Xinje XDPPro project, PLC1: XDC-60C4 (software 3.3 2016-01-26 内部测试:短信配置，自由格式配置)

PROGRAM Ladder

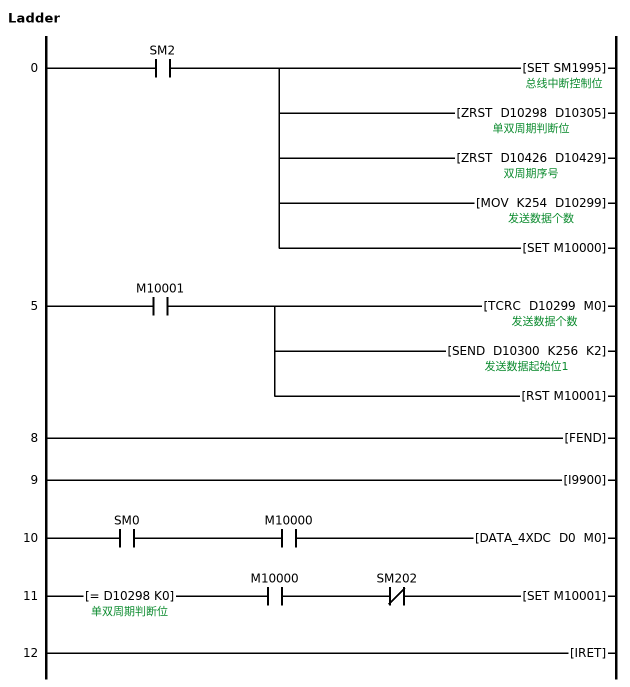
LD     SM2
SET    SM1995	; 总线中断控制位
ZRST   D10298 D10305	; 单双周期判断位
ZRST   D10426 D10429	; 双周期序号
MOV    K254 D10299	; 发送数据个数
SET    M10000
LD     M10001
TCRC   D10299 M0	; 发送数据个数
SEND   D10300 K256 K2	; 发送数据起始位1
RST    M10001
FEND
I9900
LD     SM0
AND    M10000
DATA_4XDC D0 M0
LD=    D10298 K0	; 单双周期判断位
AND    M10000
ANI    SM202
SET    M10001
IRET

COMMENTS (devices not used above)
D10301	发送数据起始位2
D10302	单周期序号
D10400	双周期数据起始位
D10554	CRC校验位
D10555	CRC校验位

C FUNCTION BLOCK data_4xdc.fcb
/*************************************************************************
   FunctionBlockName:  DATA_4XDC
   Version:            1.0.0
   Author:             cxw
   UpdateTime:         2016-1-22 15:31:37
   Comment:            
			
**************************************************************************/
void DATA_4XDC( WORD W , BIT B )
{
	#define SysRegAddr_HD_D_SD_HSD_SM
	#define offset 10300			//偏移量
	
	int i=0,j=0;
	INT16U sign=0x00ff;
	
	D[offset+0] = 0x0055;			//起始符1
	D[offset+1] = 0x0055;			//起始符2
	
	if(D[offset-2] == 0)					//单双周期判断
	{
		D[offset+2] = D[offset+126]+1;		//上周期数据序号						
		D[offset+3] = D[offset+127];
		D[offset+4] = D[offset+128];
		D[offset+5] = D[offset+129];
		
		for(i=0,j=0;i<3;i=i+1)		//轴1~3
		{
			j = i;
			D[offset+6+40*j] = (*(INT16S*)&HSD[100+20*i]&0x00ff);		//轴1位置给定
			D[offset+7+40*j] = (*(INT16S*)&HSD[100+20*i]&0xff00)>>8;
			D[offset+8+40*j] = (*(INT16S*)&HSD[101+20*i]&0x00ff);
			D[offset+9+40*j] = (*(INT16S*)&HSD[101+20*i]&0xff00)>>8;
			D[offset+10+40*j] = (*(INT16S*)&HSD[104+20*i]&0x00ff);		//轴1位置反馈
			D[offset+11+40*j] = (*(INT16S*)&HSD[104+20*i]&0xff00)>>8;
			D[offset+12+40*j] = (*(INT16S*)&HSD[105+20*i]&0x00ff);
			D[offset+13+40*j] = (*(INT16S*)&HSD[105+20*i]&0xff00)>>8;
			D[offset+14+40*j] = (*(INT16S*)&HSD[108+20*i]&0x00ff);		//轴1当前次位移脉冲数
			D[offset+15+40*j] = (*(INT16S*)&HSD[108+20*i]&0xff00)>>8;
			D[offset+16+40*j] = (*(INT16S*)&HSD[109+20*i]&0x00ff);
			D[offset+17+40*j] = (*(INT16S*)&HSD[109+20*i]&0xff00)>>8;
			
			D[offset+18+40*j] = (*(INT16S*)&SD[2012+60*i]&0x00ff);		//轴1瞬时速度给定
			D[offset+19+40*j] = (*(INT16S*)&SD[2012+60*i]&0xff00)>>8;
			D[offset+20+40*j] = (*(INT16S*)&SD[2013+60*i]&0x00ff);
			D[offset+21+40*j] = (*(INT16S*)&SD[2013+60*i]&0xff00)>>8;
			D[offset+22+40*j] = (*(INT16S*)&SD[2030+60*i]&0x00ff);		//轴1位置设定
			D[offset+23+40*j] = (*(INT16S*)&SD[2030+60*i]&0xff00)>>8;
			D[offset+24+40*j] = (*(INT16S*)&SD[2031+60*i]&0x00ff);
			D[offset+25+40*j] = (*(INT16S*)&SD[2031+60*i]&0xff00)>>8;
			D[offset+26+40*j] = (*(INT16S*)&SD[2032+60*i]&0x00ff);		//轴1速度设定
			D[offset+27+40*j] = (*(INT16S*)&SD[2032+60*i]&0xff00)>>8;
			D[offset+28+40*j] = (*(INT16S*)&SD[2033+60*i]&0x00ff);
			D[offset+29+40*j] = (*(INT16S*)&SD[2033+60*i]&0xff00)>>8;
			D[offset+30+40*j] = (*(INT16S*)&SD[2034+60*i]&0x00ff);		//轴1加速时间
			D[offset+31+40*j] = (*(INT16S*)&SD[2034+60*i]&0xff00)>>8;
			D[offset+32+40*j] = (*(INT16S*)&SD[2035+60*i]&0x00ff);					
			D[offset+33+40*j] = (*(INT16S*)&SD[2035+60*i]&0xff00)>>8;
			D[offset+34+40*j] = (*(INT16S*)&SD[2036+60*i]&0x00ff);		//轴1减速时间
			D[offset+35+40*j] = (*(INT16S*)&SD[2036+60*i]&0xff00)>>8;
			D[offset+36+40*j] = (*(INT16S*)&SD[2037+60*i]&0x00ff);					
			D[offset+37+40*j] = (*(INT16S*)&SD[2037+60*i]&0xff00)>>8;
			D[offset+38+40*j] = (*(INT16S*)&SD[2002+60*i]&0x00ff);		//轴1错误代码
			D[offset+39+40*j] = (*(INT16S*)&SD[2003+60*i]&0xff00)>>8;
			
			D[offset+40+40*j] = ((INT16U)SM[2000+20*i]);				//轴1使能标志
			D[offset+41+40*j] = ((INT16U)SM[2001+20*i]);				//轴1正在运动标志
			D[offset+42+40*j] = ((INT16U)SM[2003+20*i]);				//轴1指令完成标志
			D[offset+43+40*j] = ((INT16U)SM[2004+20*i]);				//轴1错误标志
			D[offset+44+40*j] = ((INT16U)SM[2010+20*i]);				//轴1使能控制位
			D[offset+45+40*j] = sign;
		}
		D[offset-2] = D[offset-2]+1;			
	}
	else
	{
		D[offset+126] = D[offset+2]+1;			//上周期数据序号
		if(D[offset+126]>=256)
		{
			D[offset+126] = 0;
			D[offset+127] = D[offset+127]+1;
		}
		if(D[offset+127]>=256)
		{
			D[offset+127] = 0;
			D[offset+128] = D[offset+128]+1;
		}
		if(D[offset+128]>=256)
		{
			D[offset+128] = 0;
			D[offset+129] = D[offset+129]+1;
		}
		if(D[offset+129]>=256)
		{
			D[offset+129] = 0;
		}
		
		for(i=0,j=0;i<3;i++)
		{
			j = i;
			D[offset+130+40*j] = (*(INT16S*)&HSD[100+20*i]&0x00ff);		//轴1位置给定
			D[offset+131+40*j] = (*(INT16S*)&HSD[100+20*i]&0xff00)>>8;
			D[offset+132+40*j] = (*(INT16S*)&HSD[101+20*i]&0x00ff);
			D[offset+133+40*j] = (*(INT16S*)&HSD[101+20*i]&0xff00)>>8;
			D[offset+134+40*j] = (*(INT16S*)&HSD[104+20*i]&0x00ff);		//轴1位置反馈
			D[offset+135+40*j] = (*(INT16S*)&HSD[104+20*i]&0xff00)>>8;
			D[offset+136+40*j] = (*(INT16S*)&HSD[105+20*i]&0x00ff);
			D[offset+137+40*j] = (*(INT16S*)&HSD[105+20*i]&0xff00)>>8;
			D[offset+138+40*j] = (*(INT16S*)&HSD[108+20*i]&0x00ff);		//轴1当前次位移脉冲数
			D[offset+139+40*j] = (*(INT16S*)&HSD[108+20*i]&0xff00)>>8;
			D[offset+140+40*j] = (*(INT16S*)&HSD[109+20*i]&0x00ff);
			D[offset+141+40*j] = (*(INT16S*)&HSD[109+20*i]&0xff00)>>8;
			
			D[offset+142+40*j] = (*(INT16S*)&SD[2012+60*i]&0x00ff);		//轴1瞬时速度给定
			D[offset+143+40*j] = (*(INT16S*)&SD[2012+60*i]&0xff00)>>8;
			D[offset+144+40*j] = (*(INT16S*)&SD[2013+60*i]&0x00ff);
			D[offset+145+40*j] = (*(INT16S*)&SD[2013+60*i]&0xff00)>>8;
			D[offset+146+40*j] = (*(INT16S*)&SD[2030+60*i]&0x00ff);		//轴1位置设定
			D[offset+147+40*j] = (*(INT16S*)&SD[2030+60*i]&0xff00)>>8;
			D[offset+148+40*j] = (*(INT16S*)&SD[2031+60*i]&0x00ff);
			D[offset+149+40*j] = (*(INT16S*)&SD[2031+60*i]&0xff00)>>8;
			D[offset+150+40*j] = (*(INT16S*)&SD[2032+60*i]&0x00ff);		//轴1速度设定
			D[offset+151+40*j] = (*(INT16S*)&SD[2032+60*i]&0xff00)>>8;
			D[offset+152+40*j] = (*(INT16S*)&SD[2033+60*i]&0x00ff);
			D[offset+153+40*j] = (*(INT16S*)&SD[2033+60*i]&0xff00)>>8;
			D[offset+154+40*j] = (*(INT16S*)&SD[2034+60*i]&0x00ff);		//轴1加速时间
			D[offset+155+40*j] = (*(INT16S*)&SD[2034+60*i]&0xff00)>>8;
			D[offset+156+40*j] = (*(INT16S*)&SD[2035+60*i]&0x00ff);					
			D[offset+157+40*j] = (*(INT16S*)&SD[2035+60*i]&0xff00)>>8;
			D[offset+158+40*j] = (*(INT16S*)&SD[2036+60*i]&0x00ff);		//轴1减速时间
			D[offset+159+40*j] = (*(INT16S*)&SD[2036+60*i]&0xff00)>>8;
			D[offset+160+40*j] = (*(INT16S*)&SD[2037+60*i]&0x00ff);					
			D[offset+161+40*j] = (*(INT16S*)&SD[2037+60*i]&0xff00)>>8;
			D[offset+162+40*j] = (*(INT16S*)&SD[2002+60*i]&0x00ff);		//轴1错误代码
			D[offset+163+40*j] = (*(INT16S*)&SD[2003+60*i]&0xff00)>>8;
			
			D[offset+164+40*j] = ((INT16U)SM[2000+20*i]);				//轴1使能标志
			D[offset+165+40*j] = ((INT16U)SM[2001+20*i]);				//轴1正在运动标志
			D[offset+166+40*j] = ((INT16U)SM[2003+20*i]);				//轴1指令完成标志
			D[offset+167+40*j] = ((INT16U)SM[2004+20*i]);				//轴1错误标志
			D[offset+168+40*j] = ((INT16U)SM[2010+20*i]);				//轴1使能控制位
			D[offset+169+40*j] = sign;
		}
		D[offset-2] = 0;
	}
}

C FUNCTION BLOCK tcrc.fcb
/* CRC校验生成
数据个数(n)输入:     W[0]
数据(整数)起始地址:  W[1]
...                  ...
数据(整数)结束地址:  W[n+1]
CRC校验结果存放地址：W[n+2]
W[n+3]
例:
TCRC D0 M0
数据个数: D0=0x06
数据输入: D1=0x01, D2=0x05, D3=0x48
D4=0x00, D5=0xFF, D6=0x00
结果显示: D7=0x9B, D8=0x9A */
/*************************************************************************
   FunctionBlockName:  TCRC
   Version:            1.0.0
   Author:             无锡信捷电气股份有限公司
   UpdateTime:         2010-4-22 10:01:36
   Comment:            
			CRC校验生成  
			
			数据个数(n)输入:     W[0] 
      数据(整数)起始地址:  W[1]
      ...                  ...
      数据(整数)结束地址:  W[n+1]
      CRC校验结果存放地址：W[n+2]
                           W[n+3]  
			例:
			TCRC D0 M0
			
			数据个数: D0=0x06
      数据输入: D1=0x01, D2=0x05, D3=0x48
                D4=0x00, D5=0xFF, D6=0x00
      结果显示: D7=0x9B, D8=0x9A
**************************************************************************/
void TCRC( WORD W , BIT B )
{
	int i,j,m,n;
	unsigned int crc_reg=0xffff,k;
	for (i=0;i<W[0];i++)
	{
		crc_reg^=W[i+1];
		for(j=0;j<8;j++)
		{
			if(crc_reg&0x01)
			   crc_reg=(crc_reg>>1)^0xa001;
			else
			   crc_reg=crc_reg>>1;
		}
	}
	
	m=W[0]+1;
	n=W[0]+2;
	k=crc_reg&0xff00;
	W[n]=k>>8;
	W[m]=crc_reg&0x00ff;
}